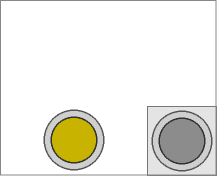
VISUALIZATION Visualization  // 217x176
    Lamp1 (39,105 70x70), variable: GVL.lamp_on, style: Lamp-Lamp1-Yellow
    PushSwitch (147,106 70x70), variable: GVL.button_pressed, behaviour: TOGGLE, style: Switch-PushSwitch-Gray
END_VISUALIZATION

(* stored: Version 1.1.0.1, ProductVersion 3.1.4024.12
   Visu Visualization: Id {3774e413-4623-487c-a752-ded68e0a8180} *)
